FUNCTION_BLOCK AM_MoveAbsolute
VAR_INPUT
	bEnable	: BOOL;
	iDistance	: INT;
	i1stRPM		: INT;
	i2ndRPM		: INT;
	i2ndSpdRange	: INT;
	iOffSetRange		: INT;
	iRatio			: REAL;
	iDtime			: INT;
	iDStep			: INT;
	MasterActualPosition	: LREAL;

END_VAR
VAR_OUTPUT
	bDone			: BOOL;
	bMoveFor		: BOOL;
	bMoveRev		: BOOL;
	iSpeedOut		: INT;



END_VAR
VAR
	RAP1: MC_ReadActualPosition;
	SpdRangeN: INT;
	SpdRangeP: INT;
	SpeedEnable: BOOL;
	OffSetN: INT;
	OffSetP: INT;
	OffSetEnable: BOOL;
	DisEn: BOOL;
	RPM1En: BOOL;
	RPM2En: BOOL;
	PosCmp1: fbServoPosCmp;
	ArmInRange: BOOL;
	RpmConvert: AM_InverterConversionHz;
	RpmConvert1: AM_InverterConversionHz;
	PosCmp2: fbServoPosCmp;
	TriggerMovFor: BOOL;
	TriggerStandStill: BOOL;
	TriggerMovRev: BOOL;
	TRIG1: R_TRIG;
	MoveEnable: BOOL;
	i1stSpeedOut : INT;
	i2ndSpeedOut : INT;
	bMoveForInt: BOOL;
	bMoveRevInt: BOOL;
	MotorMovingProfileFB: fbIndMotDecCtrl;
	PerSpd: INT;
END_VAR
VAR // added by the converter: edge detectors and wires of the graphical bodies
    _w1 : BOOL;
    _w2, _w3 : INT;
END_VAR

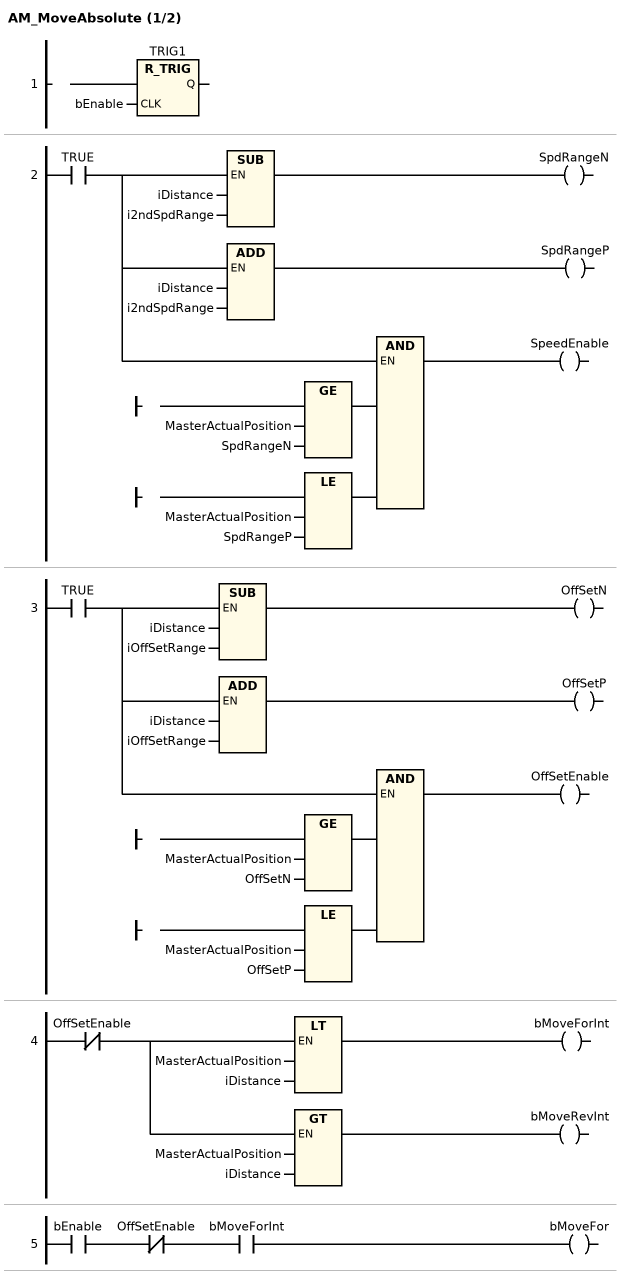
// NETWORK 1
TRIG1(CLK := bEnable); // R_TRIG

// NETWORK 2
SpdRangeN := iDistance - i2ndSpdRange;
SpdRangeP := iDistance + i2ndSpdRange;
SpeedEnable := MasterActualPosition >= SpdRangeN AND MasterActualPosition <= SpdRangeP;

// NETWORK 3
OffSetN := iDistance - iOffSetRange;
OffSetP := iDistance + iOffSetRange;
OffSetEnable := MasterActualPosition >= OffSetN AND MasterActualPosition <= OffSetP;

// NETWORK 4
_w1 := NOT OffSetEnable;
bMoveForInt := _w1 AND MasterActualPosition < iDistance;
bMoveRevInt := _w1 AND MasterActualPosition > iDistance;

// NETWORK 5
bMoveFor := bEnable AND NOT OffSetEnable AND bMoveForInt;

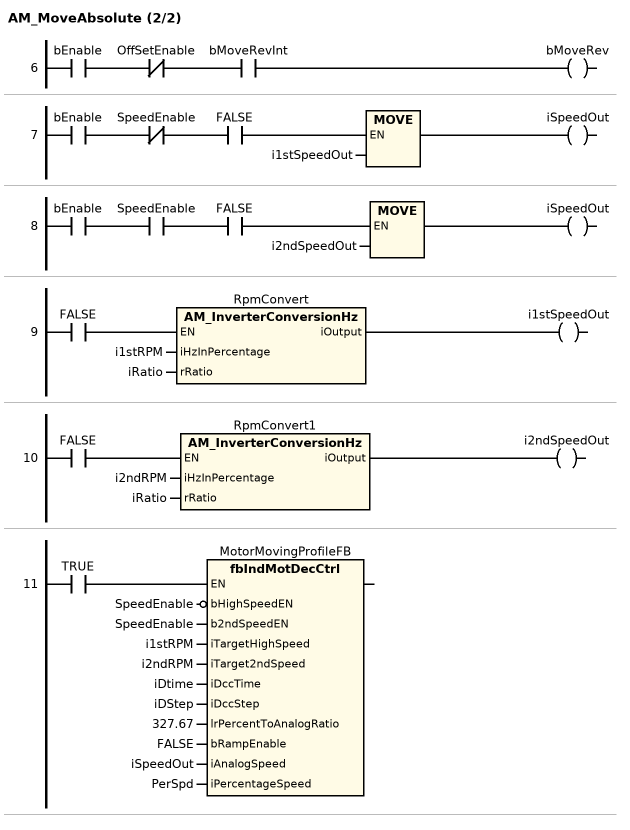
// NETWORK 6
bMoveRev := bEnable AND NOT OffSetEnable AND bMoveRevInt;

// NETWORK 7
IF bEnable AND NOT SpeedEnable AND FALSE THEN _w2 := i1stSpeedOut; END_IF
iSpeedOut := _w2;

// NETWORK 8
IF bEnable AND SpeedEnable AND FALSE THEN _w3 := i2ndSpeedOut; END_IF
iSpeedOut := _w3;

// NETWORK 9
IF FALSE THEN
    RpmConvert(iHzInPercentage := i1stRPM, rRatio := iRatio); // AM_InverterConversionHz
END_IF
i1stSpeedOut := RpmConvert.iOutput;

// NETWORK 10
IF FALSE THEN
    RpmConvert1(iHzInPercentage := i2ndRPM, rRatio := iRatio); // AM_InverterConversionHz
END_IF
i2ndSpeedOut := RpmConvert1.iOutput;

// NETWORK 11
MotorMovingProfileFB(
    bHighSpeedEN := NOT SpeedEnable,
    b2ndSpeedEN := SpeedEnable,
    iTargetHighSpeed := i1stRPM,
    iTarget2ndSpeed := i2ndRPM,
    iDccTime := iDtime,
    iDccStep := iDStep,
    lrPercentToAnalogRatio := 327.67,
    bRampEnable := FALSE,
    iAnalogSpeed := iSpeedOut,
    iPercentageSpeed := PerSpd); // fbIndMotDecCtrl

END_FUNCTION_BLOCK

(* stored: Version 1.1.0.1, ProductVersion 3.1.4024.12
   POU AM_MoveAbsolute: Id {f9106d38-7169-40bd-a732-21835203c597}, SpecialFunc None *)
